// TIA Portal V20 export
VAR_GLOBAL   // PLC tag table "Unit1"
   "BA060AZSISP201.00" AT %I700.0 : Bool;   // MAIN OP AUTO INITIATE PBL (GREEN)
   "BA060AZSISP201.01" AT %I700.1 : Bool;   // MAIN OP STOP PBL (RED)
   "BA060AZSIMP102.00" AT %I104.0 : Bool;   // LOWER 2-1 HEATER POWER TRIPPED E6168CB
   "BA060AZSIMP102.01" AT %I104.1 : Bool;   // LOWER 2-2 HEATER POWER TRIPPED E6174CB
   "BA060AZSIMP102.02" AT %I104.2 : Bool;   // LOWER 2-3 HEATER POWER TRIPPED E6180CB
   "BA060AZSIMP102.04" AT %I104.4 : Bool;   // 120VAC CONTROL POWER TR PRIMARY TRIPPED E7100CB
   "BA060AZSIMP102.05" AT %I104.5 : Bool;   // 120VAC CONTROL POWER TR SECONDARY TRIPPED E7110CB
   "BA060AZSIMP102.06" AT %I104.6 : Bool;   // CONTROL POWER ON TRIPPED E7116CB
   "BA060AZSIMP102.07" AT %I104.7 : Bool;   // MOTOR PANEL CONTROL POWER TRIPPED E7154CB
   "BA060AZSIMP102.10" AT %I105.0 : Bool;   // WEIGHT TESTER POWER STRIP OUTLET POWER TRIPPED E7160CB
   "BA060AZSIMP102.11" AT %I105.1 : Bool;   // VISION MONITOR & MCU POWER STRIP OUTLET POWER TRIPPED E7166CB
   "BA060AZSIMP102.12" AT %I105.2 : Bool;   // QR LASER MARKING TRIPPED E7172CB
   "BA060AZSIMP102.13" AT %I105.3 : Bool;   // HI-POT TESTER POWER STRIP OUTLET POWER TRIPPED E7178CB
   "BA060AZSIMP102.14" AT %I105.4 : Bool;   // FFU-1 POWER TRIPPED E7222CB
   "BA060AZSIMP102.15" AT %I105.5 : Bool;   // UPPER 1-1 TEMPERATURE CONTROLLER POWER TRIPPED E5206CB
   "BA060AZSIMP102.16" AT %I105.6 : Bool;   // UPPER 1-2 TEMPERATURE CONTROLLER POWER TRIPPED E5212CB
   "BA060AZSIMP102.17" AT %I105.7 : Bool;   // LOWER 1-1 TEMPERATURE CONTROLLER POWER TRIPPED E5218CB
   "BA060AZSIMP102.20" AT %I106.0 : Bool;   // LOWER 1-2 TEMPERATURE CONTROLLER POWER TRIPPED E5224CB
   "BA060AZSIMP102.21" AT %I106.1 : Bool;   // LOWER 1-3 TEMPERATURE CONTROLLER POWER TRIPPED E5230CB
   "BA060AZSIMP102.22" AT %I106.2 : Bool;   // UPPER 2-1 TEMPERATURE CONTROLLER POWER TRIPPED E6206CB
   "BA060AZSIMP102.23" AT %I106.3 : Bool;   // UPPER 2-2 TEMPERATURE CONTROLLER POWER TRIPPED E6212CB
   "BA060AZSIMP102.24" AT %I106.4 : Bool;   // LOWER 2-1 TEMPERATURE CONTROLLER POWER TRIPPED E6218CB
   "BA060AZSIMP102.25" AT %I106.5 : Bool;   // LOWER 2-2 TEMPERATURE CONTROLLER POWER TRIPPED E6224CB
   "BA060AZSIMP102.26" AT %I106.6 : Bool;   // LOWER 2-3 TEMPERATURE CONTROLLER POWER TRIPPED E6230CB
   "BA060AZSIMP102.30" AT %I107.0 : Bool;   // CONTROL POWER SMPS DC OK E8104PWS
   "BA060AZSIMP102.31" AT %I107.1 : Bool;   // ET200MP I/O OUTPUT POWER TRIPPED E8154CB
   "BA060AZSIMP102.32" AT %I107.2 : Bool;   // JUNCTION BOX CONTROL POWER TRIPPED E8180CB
   "BA060AZSIMP102.33" AT %I107.3 : Bool;   // CLASS 2 SMPS POWER TRIPPED E8204CB
   "BA060AZSIMP102.34" AT %I107.4 : Bool;   // CLASS 2 SMPS MONITORING E8206PWS
   "BA060AZSIMP102.35" AT %I107.5 : Bool;   // ET200ECO PN-1 POWER TRIPPED E8220CB
   "BA060AZSIMP102.36" AT %I107.6 : Bool;   // ET200ECO PN-2 POWER TRIPPED E8224CB
   "BA060AZSIMP102.37" AT %I107.7 : Bool;   // ET200ECO PN-3 POWER TRIPPED E8228CB
   "BA060AZSIMP103.00" AT %I108.0 : Bool;   // ET200ECO PN-4 POWER TRIPPED E8232CB
   "BA060AZSIMP103.01" AT %I108.1 : Bool;   // PANEL FAN POWER TRIPPED E8304CB
   "BA060AZSIMP103.03" AT %I108.3 : Bool;   // CONTROLLER POWER SMPS DC OK E8404PWS
   "BA060AZSIMP103.04" AT %I108.4 : Bool;   // CONTROLLER DC POWER TRIPPED E8406CB
   "BA060AZSIMP103.05" AT %I108.5 : Bool;   // KISTLER CONTROL POWER TRIPPED E8416CB
   "BA060AZSIMP103.06" AT %I108.6 : Bool;   // MANIFOLD-1 POWER TRIPPED E8422CB
   "BA060AZSIMP103.07" AT %I108.7 : Bool;   // MANIFOLD-2 POWER TRIPPED E8430CB
   "BA060AZSIMP103.10" AT %I109.0 : Bool;   // QR READER POWER TRIPPED E8456CB
   "BA060AZSIMP103.11" AT %I109.1 : Bool;   // QR READER POWER TRIPPED E8462CB
   "BA060AZSIMP103.12" AT %I109.2 : Bool;   // HANDY QR READER POWER TRIPPED E8468CB
   "BA060AZSIMP103.13" AT %I109.3 : Bool;   // PROFINET CONVERTER POWER TRIPPED E8474CB
   "BA060AZSIMP103.14" AT %I109.4 : Bool;   // MONITORING RELAY POWER TRIPPED E8504CB
   "BA060AZSIMP103.16" AT %I109.6 : Bool;   // SAFETY POWER SMPS DC OK E8704PWS
   "BA060AZSIMP103.17" AT %I109.7 : Bool;   // SAFETY DC POWER TRIPPED E8706CB
   "BA060AZSIMP103.20" AT %I110.0 : Bool;   // ET200SP I/O SAFETY POWER TRIPPED E8716CB
   "BA060AZSIMP103.21" AT %I110.1 : Bool;   // JUNCTION BOX CONTROL POWER TRIPPED E8736CB
   "BA060AZSIMP103.22" AT %I110.2 : Bool;   // ET200ECO PN SAFETYT-1 POWER TRIPPED E8756CB
   "BA060AZSIMP103.25" AT %I110.5 : Bool;   // CONTROL POWER SMPS DC OK E8804PWS
   "BA060AZSIMP103.26" AT %I110.6 : Bool;   // CONTROL DC POWER TRIPPED E8806CB
   "BA060AZSIMP103.27" AT %I110.7 : Bool;   // JUNCTION BOX CONTROL POWER TRIPPED E8816CB
   "BA060AZSIMP103.30" AT %I111.0 : Bool;   // DRIVE-CLIQ HUB POWER TRIPPED E8822CB
   "BA060AZSIMP103.31" AT %I111.1 : Bool;   // EQUIPMENT LED POWER TRIPPED E8828CB
   "BA060AZSICU1.Telegram_In" AT %I5000.0 : "LPD_typePDTel390In";
   "BA060AZSICU2.Telegram_In" AT %I5004.0 : "LPD_typePDTel390In";
   "BA060AZSICU3.Telegram_In" AT %I5008.0 : "LPD_typePDTel390In";
   "BA060AZSICU4.Telegram_In" AT %I5012.0 : "LPD_typePDTel390In";
   "BA060AZSISP501.00" AT %I3000.0 : Bool;   // SPARE
   "BA060AZSISP501.01" AT %I3000.1 : Bool;   // SAFETY DC POWER TRIPPED E218CB
   "BA060AZSISP501.02" AT %I3000.2 : Bool;   // CLASS 2 SMPS POWER TRIPPED E308CB
   "BA060AZSISP501.03" AT %I3000.3 : Bool;   // CLASS 2 SMPS MONITORING E310PWS
   "BA060AZSISP501.04" AT %I3000.4 : Bool;   // ET200ECO PN-1 POWER TRIPPED E324CB
   "BA060AZSISP501.05" AT %I3000.5 : Bool;   // ET200ECO PN-2 POWER TRIPPED E328CB
   "BA060AZSISP501.06" AT %I3000.6 : Bool;   // ET200ECO PN-3 POWER TRIPPED E332CB
   "BA060AZSISP501.07" AT %I3000.7 : Bool;   // ET200ECO PN-4 POWER TRIPPED E336CB
   "BA060AZSIMP101.00" AT %I100.0 : Bool;   // KISTLER 100KN PRESS POWER TRIPPED E202CB
   "BA060AZSIMP101.01" AT %I100.1 : Bool;   // KISTLER 100KN PRESS POWER TRIPPED E208CB
   "BA060AZSIMP101.02" AT %I100.2 : Bool;   // KISTLER 30KN PRESS POWER TRIPPED E214CB
   "BA060AZSIMP101.05" AT %I100.5 : Bool;   // E8404PWS CONTROLLER POWER SMPS AC POWER TRIPPED E320CB
   "BA060AZSIMP101.06" AT %I100.6 : Bool;   // E8704PWS SAFETY POWER SMPS AC POWER TRIPPED E326CB
   "BA060AZSIMP101.07" AT %I100.7 : Bool;   // E8804PWS CONTRL POWER SMPS AC POWER TRIPPED E332CB
   "BA060AZSIMP101.10" AT %I101.0 : Bool;   // PROCESSOR POWER ON TIPPRED E4120CB
   "BA060AZSIMP101.11" AT %I101.1 : Bool;   // PROGRAMING POWER OUTLET TRPPED E4126CB
   "BA060AZSIMP101.13" AT %I101.3 : Bool;   // PANEL LED POWER TRIPPED E4304CB
   "BA060AZSIMP101.15" AT %I101.5 : Bool;   // PLC POWER SMPS DC OK E4404PWS
   "BA060AZSIMP101.16" AT %I101.6 : Bool;   // CONTROL LEVEL HUB POWER TRIPPED E4420CB
   "BA060AZSIMP101.17" AT %I101.7 : Bool;   // MAIN HMI POWER TRIPPED E4426CB
   "BA060AZSIMP101.20" AT %I102.0 : Bool;   // PORTABLE HMI POWER TIPPED E4432CB
   "BA060AZSIMP101.21" AT %I102.1 : Bool;   // PORTABLE HMI POWER TIPPED E4456CB
   "BA060AZSIMP101.22" AT %I102.2 : Bool;   // 120VAC HEATER-1 POWER TR PRIMARY TRIPPED E5100CB
   "BA060AZSIMP101.25" AT %I102.5 : Bool;   // UPPER 1-1 HEATER POWER TRIPPED E5156CB
   "BA060AZSIMP101.26" AT %I102.6 : Bool;   // UPPER 1-2 HEATER POWER TRIPPED E5162CB
   "BA060AZSIMP101.27" AT %I102.7 : Bool;   // LOWER 1-1 HEATER POWER TRIPPED E5168CB
   "BA060AZSIMP101.30" AT %I103.0 : Bool;   // LOWER 1-2 HEATER POWER TRIPPED E5174CB
   "BA060AZSIMP101.31" AT %I103.1 : Bool;   // LOWER 1-3 HEATER POWER TRIPPED E5180CB
   "BA060AZSIMP101.33" AT %I103.3 : Bool;   // 120VAC HEATER-2 POWER TR PRIMARY TRIPPED E6100CB
   "BA060AZSIMP101.36" AT %I103.6 : Bool;   // UPPER 2-1 HEATER POWER TRIPPED E6156CB
   "BA060AZSIMP101.37" AT %I103.7 : Bool;   // UPPER 2-2 HEATER POWER TRIPPED E6162CB
   "BA060AZSIMP103.23" AT %I110.3 : Bool;   // ET200ECO PN SAFETYT-2 POWER TRIPPED E8762CB
   "BA060AZSISP201.10" AT %I701.0 : Bool;   // MAIN HMI POWER TRIPPED E110CB
   "BA060AZSIMP101.03" AT %I100.3 : Bool;   // SPARE
   "BA060AZSIMP101.04" AT %I100.4 : Bool;   // SPARE
   "BA060AZSIMP101.12" AT %I101.2 : Bool;   // SPARE
   "BA060AZSIMP101.14" AT %I101.4 : Bool;   // SPARE
   "BA060AZSIMP101.23" AT %I102.3 : Bool;   // SPARE
   "BA060AZSIMP101.24" AT %I102.4 : Bool;   // SPARE
   "BA060AZSIMP101.32" AT %I103.2 : Bool;   // SPARE
   "BA060AZSIMP101.34" AT %I103.4 : Bool;   // SPARE
   "BA060AZSIMP101.35" AT %I103.5 : Bool;   // SPARE
   "BA060AZSIMP102.03" AT %I104.3 : Bool;   // VISION LIGHT CONTROLLER POWER STRIP OUTLET POWER TRIPPED E7184CB
   "BA060AZSIMP102.27" AT %I106.7 : Bool;   // SPARE
   "BA060AZSIMP103.02" AT %I108.2 : Bool;   // SPARE
   "BA060AZSIMP103.15" AT %I109.5 : Bool;   // SPARE
   "BA060AZSIMP103.24" AT %I110.4 : Bool;   // SPARE
   "BA060AZSISP201.02" AT %I700.2 : Bool;   // SPARE
   "BA060AZSISP201.03" AT %I700.3 : Bool;   // SPARE
   "BA060AZSISP201.04" AT %I700.4 : Bool;   // SPARE
   "BA060AZSISP201.05" AT %I700.5 : Bool;   // SPARE
   "BA060AZSISP201.06" AT %I700.6 : Bool;   // SPARE
   "BA060AZSISP201.07" AT %I700.7 : Bool;   // SPARE
   "BA060AZSISP201.11" AT %I701.1 : Bool;   // SPARE
   "BA060AZSISP201.12" AT %I701.2 : Bool;   // SPARE
   "BA060AZSISP201.13" AT %I701.3 : Bool;   // SPARE
   "BA060AZSISP201.14" AT %I701.4 : Bool;   // SPARE
   "BA060AZSISP201.15" AT %I701.5 : Bool;   // SPARE
   "BA060AZSISP201.16" AT %I701.6 : Bool;   // SPARE
   "BA060AZSISP201.17" AT %I701.7 : Bool;   // SPARE
   "BA060ZSIBK19.06" AT %I1072.6 : Bool;   // MAIN VALVE DIGITAL PRESSURE SWITCH OUT1
   "BA060ZSIBK19.07" AT %I1072.7 : Bool;   // MAIN VALVE DIGITAL PRESSURE SWITCH OUT2
   "BA060AZSIMP103.32" AT %I111.2 : Bool;   // SPARE
   "BA060AZSIMP103.33" AT %I111.3 : Bool;   // SPARE
   "BA060AZSIMP103.34" AT %I111.4 : Bool;   // SPARE
   "BA060AZSIMP103.35" AT %I111.5 : Bool;   // SPARE
   "BA060AZSIMP103.36" AT %I111.6 : Bool;   // SPARE
   "BA060AZSIMP103.37" AT %I111.7 : Bool;   // SPARE
   "BA060AZSIMP104.00" AT %I112.0 : Bool;   // UPPER 1-1 HEATER MONITOR SIGNAL ON
   "BA060AZSIMP104.01" AT %I112.1 : Bool;   // UPPER 1-2 HEATER MONITOR SIGNAL ON
   "BA060AZSIMP104.02" AT %I112.2 : Bool;   // LOWER 1-1 HEATER MONITOR SIGNAL ON
   "BA060AZSIMP104.03" AT %I112.3 : Bool;   // LOWER 1-2 HEATER MONITOR SIGNAL ON
   "BA060AZSIMP104.04" AT %I112.4 : Bool;   // LOWER 1-3 HEATER MONITOR SIGNAL ON
   "BA060AZSIMP104.05" AT %I112.5 : Bool;   // UPPER 2-1 HEATER MONITOR SIGNAL ON
   "BA060AZSIMP104.06" AT %I112.6 : Bool;   // UPPER 2-2 HEATER MONITOR SIGNAL ON
   "BA060AZSIMP104.07" AT %I112.7 : Bool;   // LOWER 2-1 HEATER MONITOR SIGNAL ON
   "BA060AZSIMP104.10" AT %I113.0 : Bool;   // LOWER 2-2 HEATER MONITOR SIGNAL ON
   "BA060AZSIMP104.11" AT %I113.1 : Bool;   // LOWER 2-3 HEATER MONITOR SIGNAL ON
   "BA060AZSIMP104.12" AT %I113.2 : Bool;   // SPARE
   "BA060AZSIMP104.13" AT %I113.3 : Bool;   // SPARE
   "BA060AZSIMP104.14" AT %I113.4 : Bool;   // SPARE
   "BA060AZSIMP104.15" AT %I113.5 : Bool;   // SPARE
   "BA060AZSIMP104.16" AT %I113.6 : Bool;   // SPARE
   "BA060AZSIMP104.17" AT %I113.7 : Bool;   // SPARE
   "BA060AZSIMP104.20" AT %I114.0 : Bool;   // SPARE
   "BA060AZSIMP104.21" AT %I114.1 : Bool;   // SPARE
   "BA060AZSIMP104.22" AT %I114.2 : Bool;   // SPARE
   "BA060AZSIMP104.23" AT %I114.3 : Bool;   // SPARE
   "BA060AZSIMP104.24" AT %I114.4 : Bool;   // SPARE
   "BA060AZSIMP104.25" AT %I114.5 : Bool;   // SPARE
   "BA060AZSIMP104.26" AT %I114.6 : Bool;   // SPARE
   "BA060AZSIMP104.27" AT %I114.7 : Bool;   // SPARE
   "BA060AZSIMP104.30" AT %I115.0 : Bool;   // SPARE
   "BA060AZSIMP104.31" AT %I115.1 : Bool;   // SPARE
   "BA060AZSIMP104.32" AT %I115.2 : Bool;   // SPARE
   "BA060AZSIMP104.33" AT %I115.3 : Bool;   // SPARE
   "BA060AZSIMP104.34" AT %I115.4 : Bool;   // SPARE
   "BA060AZSIMP104.35" AT %I115.5 : Bool;   // SPARE
   "BA060AZSIMP104.36" AT %I115.6 : Bool;   // SPARE
   "BA060AZSIMP104.37" AT %I115.7 : Bool;   // SPARE
   "BA060AZSISP202.00" AT %Q700.0 : Bool;   // MAIN OP AUTO INITIATE PBL LAMP ON (GREEN)
   "BA060AZSISP202.01" AT %Q700.1 : Bool;   // MAIN OP STOP PBL LAMP ON (RED)
   "BA060AZSISP202.02" AT %Q700.2 : Bool;   // RESERVE
   "BA060AZSISP202.03" AT %Q700.3 : Bool;   // MAIN OP ENABLE PBL LAMP ON (WHITE)
   "BA060AZSISP202.04" AT %Q700.4 : Bool;   // MAIN OP SAFETY RESET PBL LAMP ON (BLUE)
   "BA060AZSISP202.05" AT %Q700.5 : Bool;   // SPARE
   "BA060AZSISP202.06" AT %Q700.6 : Bool;   // SPARE
   "BA060AZSISP202.07" AT %Q700.7 : Bool;   // SPARE
   "BA060AZSISP202.10" AT %Q701.0 : Bool;   // TOWER LAMP 1 ON (RED)
   "BA060AZSISP202.11" AT %Q701.1 : Bool;   // TOWER LAMP 2 ON (AMBER)
   "BA060AZSISP202.12" AT %Q701.2 : Bool;   // TOWER LAMP 3 ON (GREEN)
   "BA060AZSISP202.13" AT %Q701.3 : Bool;   // TOWER LAMP 4 ON (WHITE)
   "BA060AZSISP202.14" AT %Q701.4 : Bool;   // TOWER LAMP 5 ON (BLUE)
   "BA060AZSISP202.15" AT %Q701.5 : Bool;   // TOWER LAMP BUZZER ON
   "BA060AZSISP202.16" AT %Q701.6 : Bool;   // SPARE
   "BA060AZSISP202.17" AT %Q701.7 : Bool;   // SPARE
   "BA060AZSICU1.Telegram_out" AT %Q5000.0 : "LPD_typePDTel390Out";
   "BA060AZSICU2.Telegram_out" AT %Q5004.0 : "LPD_typePDTel390Out";
   "BA060AZSICU3.Telegram_out" AT %Q5008.0 : "LPD_typePDTel390Out";
   "BA060AZSICU4.Telegram_out" AT %Q5012.0 : "LPD_typePDTel390Out";
   "BA060AZSIMP105.10" AT %Q101.0 : Bool;   // QR MARKER TOWER LAMP 1 ON (RED)
   "BA060AZSIMP105.11" AT %Q101.1 : Bool;   // QR MARKER TOWER LAMP 2 ON (AMBER)
   "BA060AZSIMP105.12" AT %Q101.2 : Bool;   // QR MARKER TOWER LAMP 3 ON (GREEN)
   "BA060AZSIMP105.13" AT %Q101.3 : Bool;   // QR MARKER TOWER LAMP 4 ON (WHITE)
   "BA060AZSIMP105.14" AT %Q101.4 : Bool;   // QR MARKER TOWER LAMP 5 ON (BLUE)
   "BA060AZSIMP105.15" AT %Q101.5 : Bool;   // QR MARKER TOWER LAMP BUZZER ON
   "BA060AZSISP504.00" AT %Q3000.0 : Bool;   // CLASS2 SMPS ALARM RESET
   "BA060AZSISP504.01" AT %Q3000.1 : Bool;   // SPARE
   "BA060AZSIMP105.00" AT %Q100.0 : Bool;   // EQUIPMENT LED LAMP RELAY ON
   "BA060AZSIMP105.03" AT %Q100.3 : Bool;   // CLASS2 SMPS ALARM RESET
   "BA060AZSIMP105.04" AT %Q100.4 : Bool;   // SPARE
   "BA060AZSIMP105.05" AT %Q100.5 : Bool;   // SPARE
   "BA060AZSIMP105.06" AT %Q100.6 : Bool;   // SPARE
   "BA060AZSIMP105.07" AT %Q100.7 : Bool;   // SPARE
   "BA060AZSIMP105.16" AT %Q101.6 : Bool;   // SPARE
   "BA060AZSIMP105.17" AT %Q101.7 : Bool;   // SPARE
   "BA060AZSIMP105.20" AT %Q102.0 : Bool;   // SPARE
   "BA060AZSIMP105.21" AT %Q102.1 : Bool;   // SPARE
   "BA060AZSIMP105.22" AT %Q102.2 : Bool;   // SPARE
   "BA060AZSIMP105.23" AT %Q102.3 : Bool;   // SPARE
   "BA060AZSIMP105.01" AT %Q100.1 : Bool;   // SPARE
   "BA060AZSIMP105.02" AT %Q100.2 : Bool;   // SPARE
   "BA060AZSIMP105.24" AT %Q102.4 : Bool;   // SPARE
   "BA060AZSIMP105.25" AT %Q102.5 : Bool;   // SPARE
   "BA060AZSIMP105.26" AT %Q102.6 : Bool;   // SPARE
   "BA060AZSIMP105.27" AT %Q102.7 : Bool;   // SPARE
   "BA060AZSIMP105.30" AT %Q103.0 : Bool;   // SPARE
   "BA060AZSIMP105.31" AT %Q103.1 : Bool;   // SPARE
   "BA060AZSIMP105.32" AT %Q103.2 : Bool;   // SPARE
   "BA060AZSIMP105.33" AT %Q103.3 : Bool;   // SPARE
   "BA060AZSIMP105.34" AT %Q103.4 : Bool;   // SPARE
   "BA060AZSIMP105.35" AT %Q103.5 : Bool;   // SPARE
   "BA060AZSIMP105.36" AT %Q103.6 : Bool;   // SPARE
   "BA060AZSIMP105.37" AT %Q103.7 : Bool;   // SPARE
END_VAR
VAR_GLOBAL CONSTANT   // user constants
   U1_NO_OF_EMs : Int := 13;   // Highest Value of equipment modules in the unit (Counting starts from 0)
   U1_EM0 : Int := 0;   // Equipment Module 0
   U1_EM1 : Int := 1;   // Equipment Module 1
   U1_EM2 : Int := 2;   // Equipment Module 2
   U1_EM3 : Int := 3;   // Equipment Module 3
   U1_EM4 : Int := 4;   // Equipment Module 4
   U1_EM5 : Int := 5;   // Equipment Module 5
   U1_EM6 : Int := 6;   // Equipment Module 6
   U1_EM7 : Int := 7;   // Equipment Module 7
   U1_EM8 : Int := 8;   // Equipment Module 8
   U1_EM9 : Int := 9;   // Equipment Module 9
   U1_EM10 : Int := 10;   // Equipment Module 10
   U1_EM11 : Int := 11;   // Equipment Module 11
   U1_EM12 : Int := 12;   // Equipment Module 12
   U1_EM13 : Int := 13;   // Equipment Module 13
END_VAR
